PROGRAM OP160_Robo_Byte_Mapping
VAR

//registerout

	OP160_Robo_IN_Byte2: BYTE_AS_BIT;
	OP160_Robo_IN_Byte3: BYTE_AS_BIT;
	OP160_Robo_IN_Byte4: BYTE_AS_BIT;
	OP160_Robo_IN_Byte5: BYTE_AS_BIT;
	OP160_Robo_IN_Byte6: BYTE_AS_BIT;
	OP160_Robo_IN_Byte7: BYTE_AS_BIT;
	OP160_Robo_IN_Byte8: BYTE_AS_BIT;
	OP160_Robo_Out_Byte1: BIT_AS_BYTE;
	OP160_Robo_Out_Byte2: BIT_AS_BYTE;
	OP160_Robo_Out_Byte3: BIT_AS_BYTE;
	OP160_Robo_Out_Byte4: BIT_AS_BYTE;
	OP160_Robo_Out_Byte5: BIT_AS_BYTE;
	OP160_Robo_Out_Byte6: BIT_AS_BYTE;
	OP160_Robo_Out_Byte7: BIT_AS_BYTE;
	OP160_Robo_Out_Byte8: BIT_AS_BYTE;
	OP160_EI_Rdy_Reject: BOOL;
END_VAR

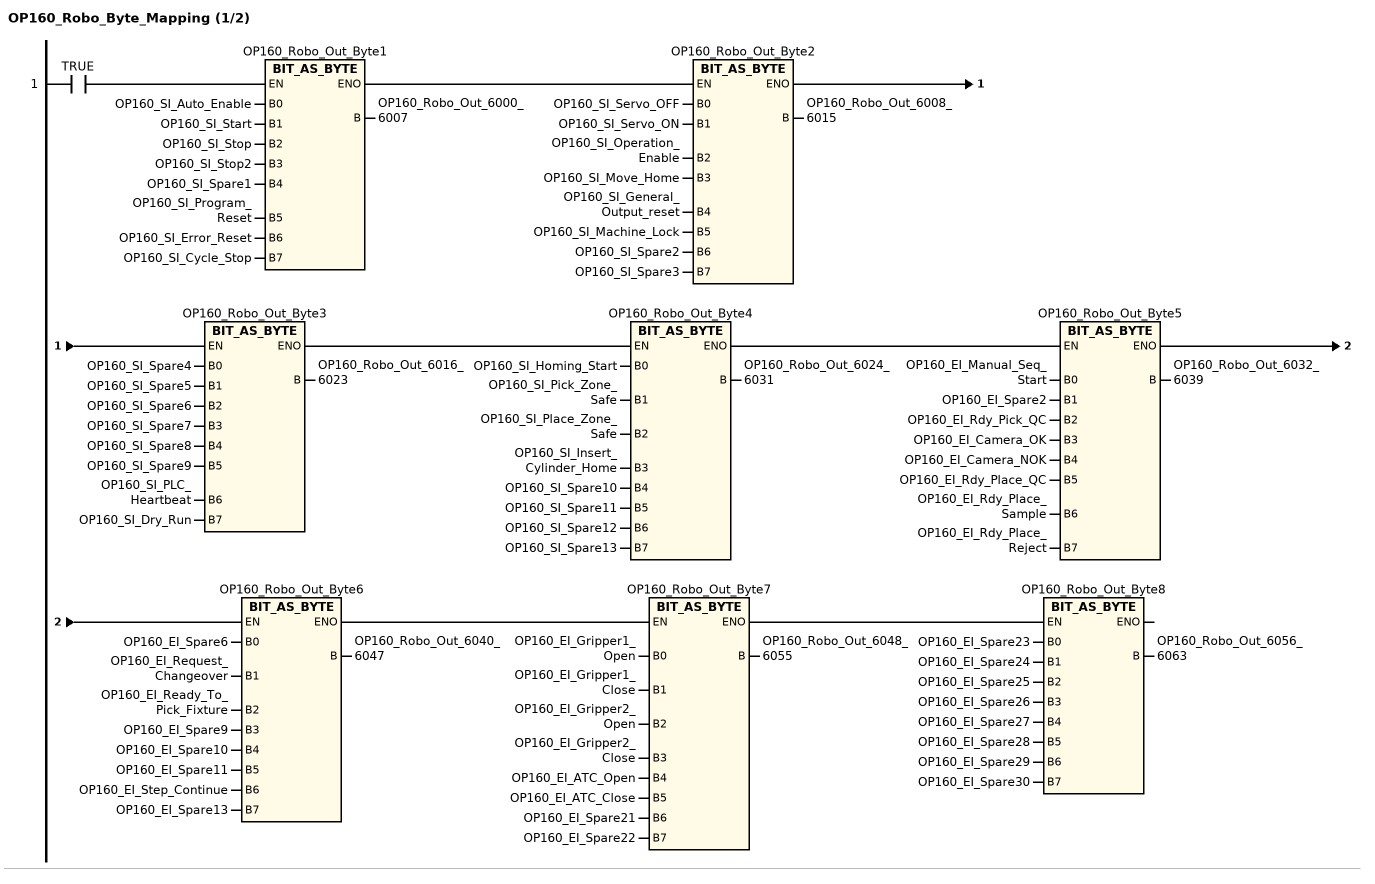
// NETWORK 1
OP160_Robo_Out_Byte1(
    B0 := OP160_SI_Auto_Enable,
    B1 := OP160_SI_Start,
    B2 := OP160_SI_Stop,
    B3 := OP160_SI_Stop2,
    B4 := OP160_SI_Spare1,
    B5 := OP160_SI_Program_Reset,
    B6 := OP160_SI_Error_Reset,
    B7 := OP160_SI_Cycle_Stop,
    B => OP160_Robo_Out_6000_6007); // BIT_AS_BYTE
OP160_Robo_Out_Byte2(
    B0 := OP160_SI_Servo_OFF,
    B1 := OP160_SI_Servo_ON,
    B2 := OP160_SI_Operation_Enable,
    B3 := OP160_SI_Move_Home,
    B4 := OP160_SI_General_Output_reset,
    B5 := OP160_SI_Machine_Lock,
    B6 := OP160_SI_Spare2,
    B7 := OP160_SI_Spare3,
    B => OP160_Robo_Out_6008_6015); // BIT_AS_BYTE
OP160_Robo_Out_Byte3(
    B0 := OP160_SI_Spare4,
    B1 := OP160_SI_Spare5,
    B2 := OP160_SI_Spare6,
    B3 := OP160_SI_Spare7,
    B4 := OP160_SI_Spare8,
    B5 := OP160_SI_Spare9,
    B6 := OP160_SI_PLC_Heartbeat,
    B7 := OP160_SI_Dry_Run,
    B => OP160_Robo_Out_6016_6023); // BIT_AS_BYTE
OP160_Robo_Out_Byte4(
    B0 := OP160_SI_Homing_Start,
    B1 := OP160_SI_Pick_Zone_Safe,
    B2 := OP160_SI_Place_Zone_Safe,
    B3 := OP160_SI_Insert_Cylinder_Home,
    B4 := OP160_SI_Spare10,
    B5 := OP160_SI_Spare11,
    B6 := OP160_SI_Spare12,
    B7 := OP160_SI_Spare13,
    B => OP160_Robo_Out_6024_6031); // BIT_AS_BYTE
OP160_Robo_Out_Byte5(
    B0 := OP160_EI_Manual_Seq_Start,
    B1 := OP160_EI_Spare2,
    B2 := OP160_EI_Rdy_Pick_QC,
    B3 := OP160_EI_Camera_OK,
    B4 := OP160_EI_Camera_NOK,
    B5 := OP160_EI_Rdy_Place_QC,
    B6 := OP160_EI_Rdy_Place_Sample,
    B7 := OP160_EI_Rdy_Place_Reject,
    B => OP160_Robo_Out_6032_6039); // BIT_AS_BYTE
OP160_Robo_Out_Byte6(
    B0 := OP160_EI_Spare6,
    B1 := OP160_EI_Request_Changeover,
    B2 := OP160_EI_Ready_To_Pick_Fixture,
    B3 := OP160_EI_Spare9,
    B4 := OP160_EI_Spare10,
    B5 := OP160_EI_Spare11,
    B6 := OP160_EI_Step_Continue,
    B7 := OP160_EI_Spare13,
    B => OP160_Robo_Out_6040_6047); // BIT_AS_BYTE
OP160_Robo_Out_Byte7(
    B0 := OP160_EI_Gripper1_Open,
    B1 := OP160_EI_Gripper1_Close,
    B2 := OP160_EI_Gripper2_Open,
    B3 := OP160_EI_Gripper2_Close,
    B4 := OP160_EI_ATC_Open,
    B5 := OP160_EI_ATC_Close,
    B6 := OP160_EI_Spare21,
    B7 := OP160_EI_Spare22,
    B => OP160_Robo_Out_6048_6055); // BIT_AS_BYTE
OP160_Robo_Out_Byte8(
    B0 := OP160_EI_Spare23,
    B1 := OP160_EI_Spare24,
    B2 := OP160_EI_Spare25,
    B3 := OP160_EI_Spare26,
    B4 := OP160_EI_Spare27,
    B5 := OP160_EI_Spare28,
    B6 := OP160_EI_Spare29,
    B7 := OP160_EI_Spare30,
    B => OP160_Robo_Out_6056_6063); // BIT_AS_BYTE

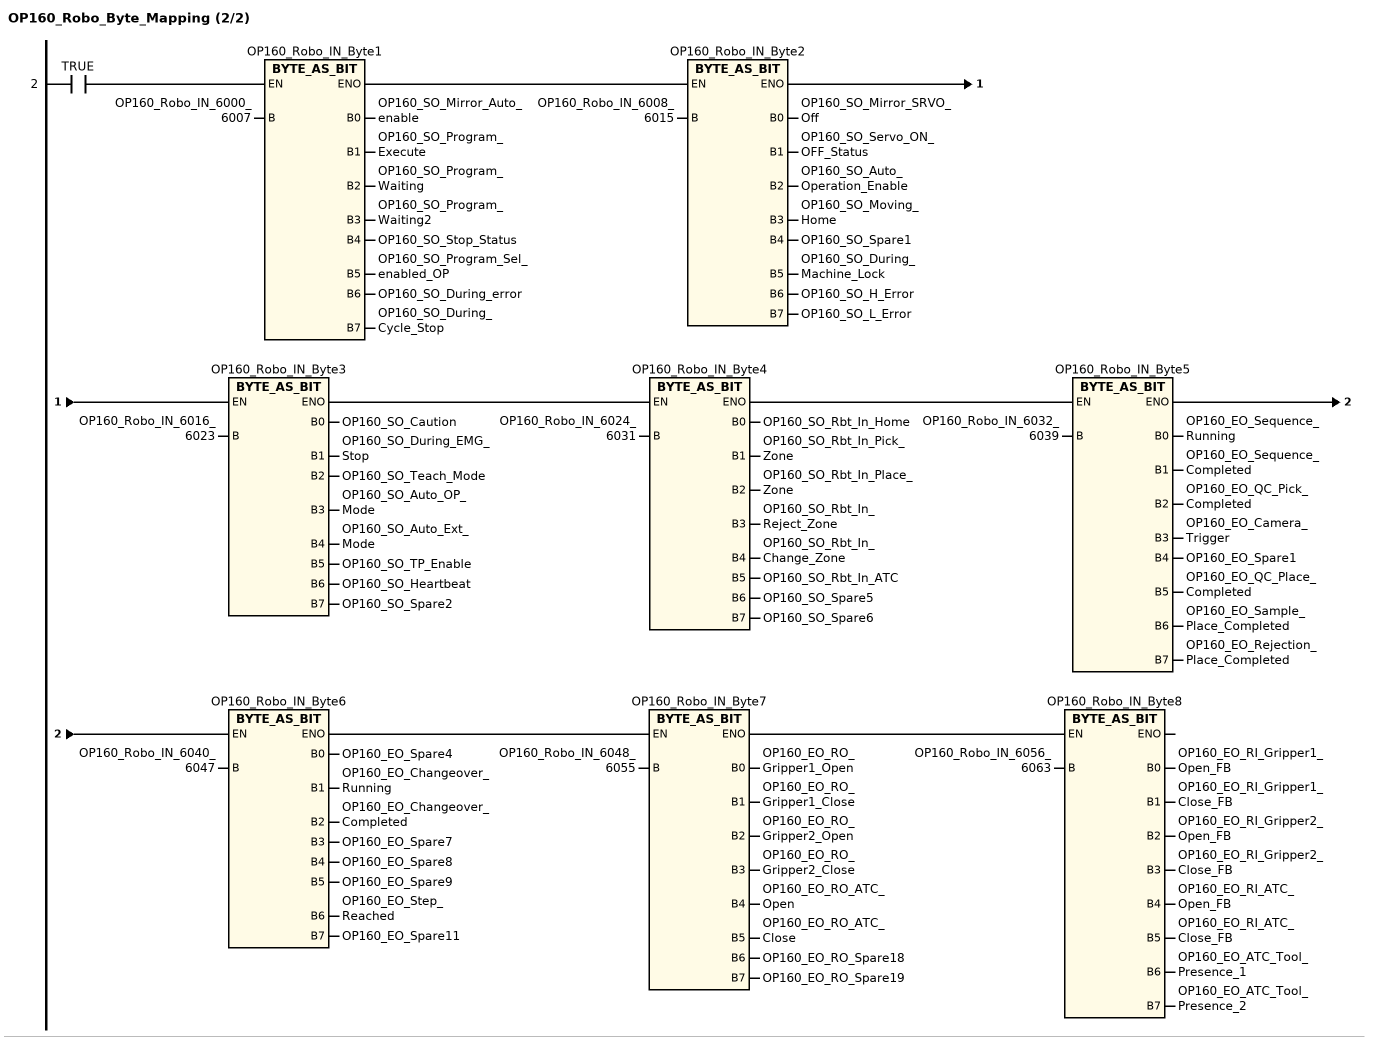
// NETWORK 2
OP160_Robo_IN_Byte1(
    B := OP160_Robo_IN_6000_6007,
    B0 => OP160_SO_Mirror_Auto_enable,
    B1 => OP160_SO_Program_Execute,
    B2 => OP160_SO_Program_Waiting,
    B3 => OP160_SO_Program_Waiting2,
    B4 => OP160_SO_Stop_Status,
    B5 => OP160_SO_Program_Sel_enabled_OP,
    B6 => OP160_SO_During_error,
    B7 => OP160_SO_During_Cycle_Stop); // BYTE_AS_BIT
OP160_Robo_IN_Byte2(
    B := OP160_Robo_IN_6008_6015,
    B0 => OP160_SO_Mirror_SRVO_Off,
    B1 => OP160_SO_Servo_ON_OFF_Status,
    B2 => OP160_SO_Auto_Operation_Enable,
    B3 => OP160_SO_Moving_Home,
    B4 => OP160_SO_Spare1,
    B5 => OP160_SO_During_Machine_Lock,
    B6 => OP160_SO_H_Error,
    B7 => OP160_SO_L_Error); // BYTE_AS_BIT
OP160_Robo_IN_Byte3(
    B := OP160_Robo_IN_6016_6023,
    B0 => OP160_SO_Caution,
    B1 => OP160_SO_During_EMG_Stop,
    B2 => OP160_SO_Teach_Mode,
    B3 => OP160_SO_Auto_OP_Mode,
    B4 => OP160_SO_Auto_Ext_Mode,
    B5 => OP160_SO_TP_Enable,
    B6 => OP160_SO_Heartbeat,
    B7 => OP160_SO_Spare2); // BYTE_AS_BIT
OP160_Robo_IN_Byte4(
    B := OP160_Robo_IN_6024_6031,
    B0 => OP160_SO_Rbt_In_Home,
    B1 => OP160_SO_Rbt_In_Pick_Zone,
    B2 => OP160_SO_Rbt_In_Place_Zone,
    B3 => OP160_SO_Rbt_In_Reject_Zone,
    B4 => OP160_SO_Rbt_In_Change_Zone,
    B5 => OP160_SO_Rbt_In_ATC,
    B6 => OP160_SO_Spare5,
    B7 => OP160_SO_Spare6); // BYTE_AS_BIT
OP160_Robo_IN_Byte5(
    B := OP160_Robo_IN_6032_6039,
    B0 => OP160_EO_Sequence_Running,
    B1 => OP160_EO_Sequence_Completed,
    B2 => OP160_EO_QC_Pick_Completed,
    B3 => OP160_EO_Camera_Trigger,
    B4 => OP160_EO_Spare1,
    B5 => OP160_EO_QC_Place_Completed,
    B6 => OP160_EO_Sample_Place_Completed,
    B7 => OP160_EO_Rejection_Place_Completed); // BYTE_AS_BIT
OP160_Robo_IN_Byte6(
    B := OP160_Robo_IN_6040_6047,
    B0 => OP160_EO_Spare4,
    B1 => OP160_EO_Changeover_Running,
    B2 => OP160_EO_Changeover_Completed,
    B3 => OP160_EO_Spare7,
    B4 => OP160_EO_Spare8,
    B5 => OP160_EO_Spare9,
    B6 => OP160_EO_Step_Reached,
    B7 => OP160_EO_Spare11); // BYTE_AS_BIT
OP160_Robo_IN_Byte7(
    B := OP160_Robo_IN_6048_6055,
    B0 => OP160_EO_RO_Gripper1_Open,
    B1 => OP160_EO_RO_Gripper1_Close,
    B2 => OP160_EO_RO_Gripper2_Open,
    B3 => OP160_EO_RO_Gripper2_Close,
    B4 => OP160_EO_RO_ATC_Open,
    B5 => OP160_EO_RO_ATC_Close,
    B6 => OP160_EO_RO_Spare18,
    B7 => OP160_EO_RO_Spare19); // BYTE_AS_BIT
OP160_Robo_IN_Byte8(
    B := OP160_Robo_IN_6056_6063,
    B0 => OP160_EO_RI_Gripper1_Open_FB,
    B1 => OP160_EO_RI_Gripper1_Close_FB,
    B2 => OP160_EO_RI_Gripper2_Open_FB,
    B3 => OP160_EO_RI_Gripper2_Close_FB,
    B4 => OP160_EO_RI_ATC_Open_FB,
    B5 => OP160_EO_RI_ATC_Close_FB,
    B6 => OP160_EO_ATC_Tool_Presence_1,
    B7 => OP160_EO_ATC_Tool_Presence_2); // BYTE_AS_BIT

END_PROGRAM

(* stored: Version 1.1.0.1, ProductVersion 3.1.4024.11
   POU OP160_Robo_Byte_Mapping: Id {ee12f2f5-a400-43ab-9b87-eb48eeae12b0}, SpecialFunc None *)
